{attribute 'GeneratedUsingTerminal: EL3692-0000-0020'}
{attribute addProperty BoxType "EL3692-0000-0020"}
{attribute addProperty Id "ModeBYTE1RangeSINT1"}
{attribute addProperty CRC "616581440"}
{attribute addProperty Size "2"}
TYPE Settings_24C04940 :
STRUCT
	{attribute addProperty Name "Mode"}
	Mode : BYTE;
	{attribute addProperty Name "Range"}
	Range : SINT;
END_STRUCT
END_TYPE

(* stored: Version 1.2.0.0, ProductVersion 3.1.4024.11
   DUT Settings_24C04940: Id {39381916-4e47-0980-0a46-a76905b1bd13} *)
